LIN {X 0,Y 277.777,Z 1042.404,A -85,B 0,C 180,E1 8080.573,E2 8080.573} C_VEL
LIN {X 0,Y 260.235,Z 1059.705,A -85,B 0,C 180,E1 8078.402,E2 8078.402} C_VEL
LIN {X 0,Y 244.784,Z 1073.617,A -85,B 0,C 180,E1 8076.2,E2 8076.2} C_VEL
LIN {X 0,Y 227.244,Z 1088.097,A -85,B 0,C 180,E1 8073.276,E2 8073.276} C_VEL
LIN {X 0,Y 207.963,Z 1102.365,A -85,B 0,C 180,E1 8069.385,E2 8069.385} C_VEL
LIN {X 0,Y 192.676,Z 1112.751,A -85,B 0,C 180,E1 8065.598,E2 8065.598} C_VEL
LIN {X 0,Y 177.571,Z 1122.315,A -85,B 0,C 180,E1 8060.99,E2 8060.99} C_VEL
LIN {X 0,Y 159.969,Z 1132.7,A -85,B 0,C 180,E1 8053.93,E2 8053.93} C_VEL
LIN {X 0,Y 147.003,Z 1139.922,A -85,B 0,C 180,E1 8046.765,E2 8046.765} C_VEL
LIN {X 0,Y 137.193,Z 1145.374,A -85,B 0,C 180,E1 8039.228,E2 8039.228} C_VEL
LIN {X 0,Y 128.774,Z 1150.343,A -85,B 0,C 180,E1 8029.504,E2 8029.504} C_VEL
LIN {X 0,Y 123.283,Z 1154.147,A -85,B 0,C 180,E1 8017.925,E2 8017.925} C_VEL
LIN {X 0,Y 121.496,Z 1156.08,A -85,B 0,C 180,E1 8008.585,E2 8008.585} C_VEL
LIN {X 0,Y 121.206,Z 1157.152,A -85,B 0,C 180,E1 8000.024,E2 8000.024} C_VEL
LIN {X 0,Y 121.981,Z 1157.579,A -85,B 0,C 180,E1 7990.86,E2 7990.86} C_VEL
LIN {X 0,Y 124.84,Z 1157.139,A -85,B 0,C 180,E1 7980.754,E2 7980.754} C_VEL
LIN {X 0,Y 130.177,Z 1155.784,A -85,B 0,C 180,E1 7971.527,E2 7971.527} C_VEL
LIN {X 0,Y 138.594,Z 1153.323,A -85,B 0,C 180,E1 7962.62,E2 7962.62} C_VEL
LIN {X 0,Y 152.039,Z 1149.022,A -85,B 0,C 180,E1 7953.364,E2 7953.364} C_VEL
LIN {X 0,Y 168.555,Z 1142.861,A -85,B 0,C 180,E1 7945.623,E2 7945.623} C_VEL
LIN {X 0,Y 183.712,Z 1136.651,A -85,B 0,C 180,E1 7940.385,E2 7940.385} C_VEL
LIN {X 0,Y 201.418,Z 1128.646,A -85,B 0,C 180,E1 7935.627,E2 7935.627} C_VEL
LIN {X 0,Y 223.132,Z 1117.531,A -85,B 0,C 180,E1 7931.085,E2 7931.085} C_VEL
LIN {X 0,Y 241.336,Z 1107.052,A -85,B 0,C 180,E1 7928.035,E2 7928.035} C_VEL
LIN {X 0,Y 259.171,Z 1095.723,A -85,B 0,C 180,E1 7925.532,E2 7925.532} C_VEL
LIN {X 0,Y 280.353,Z 1080.74,A -85,B 0,C 180,E1 7923.031,E2 7923.031} C_VEL
LIN {X 0,Y 299.018,Z 1065.79,A -85,B 0,C 180,E1 7921.149,E2 7921.149} C_VEL
LIN {X 0,Y 314.959,Z 1051.738,A -85,B 0,C 180,E1 7919.738,E2 7919.738} C_VEL
LIN {X 0,Y 331.272,Z 1035.907,A -85,B 0,C 180,E1 7918.443,E2 7918.443} C_VEL
LIN {X 0,Y 336.652,Z 1030.337,A -85,B 0,C 180,E1 7918.031,E2 7918.031} C_VEL
LIN {X 0,Y 326.224,Z 1041.38,A -85,B 0,C 180,E1 7917.323,E2 7917.323} C_VEL
LIN {X 0,Y 320.827,Z 1046.926,A -85,B 0,C 180,E1 7917.12,E2 7917.12} C_VEL
LIN {X 0,Y 305.219,Z 1061.315,A -85,B 0,C 180,E1 7917.168,E2 7917.168} C_VEL
LIN {X 0,Y 300.311,Z 1065.535,A -85,B 0,C 180,E1 7916.938,E2 7916.938} C_VEL
LIN {X 0,Y 283.815,Z 1079.451,A -85,B 0,C 180,E1 7915.551,E2 7915.551} C_VEL
LIN {X 0,Y 264.581,Z 1094.292,A -85,B 0,C 180,E1 7913.66,E2 7913.66} C_VEL
LIN {X 0,Y 241.035,Z 1110.559,A -85,B 0,C 180,E1 7910.847,E2 7910.847} C_VEL
LIN {X 0,Y 222,Z 1122.424,A -85,B 0,C 180,E1 7908.043,E2 7908.043} C_VEL
LIN {X 0,Y 203.24,Z 1133.159,A -85,B 0,C 180,E1 7904.632,E2 7904.632} C_VEL
LIN {X 0,Y 180.343,Z 1145.085,A -85,B 0,C 180,E1 7899.216,E2 7899.216} C_VEL
LIN {X 0,Y 162.143,Z 1153.663,A -85,B 0,C 180,E1 7893.399,E2 7893.399} C_VEL
LIN {X 0,Y 146.993,Z 1160.411,A -85,B 0,C 180,E1 7886.789,E2 7886.789} C_VEL
LIN {X 0,Y 131.975,Z 1166.918,A -85,B 0,C 180,E1 7877.298,E2 7877.298} C_VEL
LIN {X 0,Y 120.616,Z 1171.822,A -85,B 0,C 180,E1 7865.47,E2 7865.47} C_VEL
LIN {X 0,Y 115.084,Z 1174.558,A -85,B 0,C 180,E1 7854.647,E2 7854.647} C_VEL
LIN {X 0,Y 113.015,Z 1175.991,A -85,B 0,C 180,E1 7844.867,E2 7844.867} C_VEL
LIN {X 0,Y 112.884,Z 1176.51,A -85,B 0,C 180,E1 7836.102,E2 7836.102} C_VEL
LIN {X 0,Y 113.083,Z 1176.346,A -85,B 0,C 180,E1 7829.494,E2 7829.494} C_VEL
LIN {X 0,Y 112.893,Z 1175.456,A -85,B 0,C 180,E1 7822.366,E2 7822.366} C_VEL
LIN {X 0,Y 113.288,Z 1173.656,A -85,B 0,C 180,E1 7813.595,E2 7813.595} C_VEL
LIN {X 0,Y 115.693,Z 1170.698,A -85,B 0,C 180,E1 7803.848,E2 7803.848} C_VEL
LIN {X 0,Y 120.925,Z 1166.519,A -85,B 0,C 180,E1 7794.052,E2 7794.052} C_VEL
LIN {X 0,Y 129.84,Z 1160.665,A -85,B 0,C 180,E1 7784.262,E2 7784.262} C_VEL
LIN {X 0,Y 144.741,Z 1151.55,A -85,B 0,C 180,E1 7774.009,E2 7774.009} C_VEL
LIN {X 0,Y 158.897,Z 1142.863,A -85,B 0,C 180,E1 7767.346,E2 7767.346} C_VEL
LIN {X 0,Y 173.719,Z 1133.462,A -85,B 0,C 180,E1 7762.082,E2 7762.082} C_VEL
LIN {X 0,Y 192.717,Z 1120.731,A -85,B 0,C 180,E1 7756.891,E2 7756.891} C_VEL
LIN {X 0,Y 212.206,Z 1106.31,A -85,B 0,C 180,E1 7752.755,E2 7752.755} C_VEL
LIN {X 0,Y 228.409,Z 1093.381,A -85,B 0,C 180,E1 7749.96,E2 7749.96} C_VEL
LIN {X 0,Y 246.957,Z 1077.339,A -85,B 0,C 180,E1 7747.284,E2 7747.284} C_VEL
LIN {X 0,Y 266.154,Z 1058.803,A -85,B 0,C 180,E1 7744.957,E2 7744.957} C_VEL
LIN {X 0,Y 281.444,Z 1042.59,A -85,B 0,C 180,E1 7743.365,E2 7743.365} C_VEL
LIN {X 0,Y 296.14,Z 1025.559,A -85,B 0,C 180,E1 7742.016,E2 7742.016} C_VEL
LIN {X 0,Y 313.472,Z 1003.187,A -85,B 0,C 180,E1 7740.603,E2 7740.603} C_VEL
LIN {X 0,Y 326.96,Z 983.532,A -85,B 0,C 180,E1 7739.615,E2 7739.615} C_VEL
LIN {X 0,Y 338.52,Z 964.867,A -85,B 0,C 180,E1 7738.848,E2 7738.848} C_VEL
LIN {X 0,Y 350.134,Z 943.92,A -85,B 0,C 180,E1 7738.141,E2 7738.141} C_VEL
LIN {X 0,Y 362.303,Z 918.548,A -85,B 0,C 180,E1 7737.463,E2 7737.463} C_VEL
LIN {X 0,Y 371.204,Z 896.845,A -85,B 0,C 180,E1 7737.002,E2 7737.002} C_VEL
LIN {X 0,Y 378.593,Z 875.937,A -85,B 0,C 180,E1 7736.647,E2 7736.647} C_VEL
LIN {X 0,Y 386.321,Z 849.767,A -85,B 0,C 180,E1 7736.294,E2 7736.294} C_VEL
LIN {X 0,Y 392.167,Z 823.299,A -85,B 0,C 180,E1 7735.962,E2 7735.962} C_VEL
LIN {X 0,Y 395.874,Z 800.827,A -85,B 0,C 180,E1 7735.692,E2 7735.692} C_VEL
LIN {X 0,Y 411.944,Z 668.915,A -85,B 0,C 180,E1 7734.149,E2 7734.149} C_VEL
LIN {X 0,Y 411.886,Z 668.578,A -85,B 0,C 180,E1 7732.827,E2 7732.827} C_VEL
LIN {X 0,Y 395.068,Z 804.017,A -85,B 0,C 180,E1 7731.344,E2 7731.344} C_VEL
LIN {X 0,Y 390.125,Z 831.221,A -85,B 0,C 180,E1 7731.017,E2 7731.017} C_VEL
LIN {X 0,Y 383.915,Z 855.88,A -85,B 0,C 180,E1 7730.656,E2 7730.656} C_VEL
LIN {X 0,Y 377.386,Z 877.053,A -85,B 0,C 180,E1 7730.26,E2 7730.26} C_VEL
LIN {X 0,Y 369.182,Z 899.494,A -85,B 0,C 180,E1 7729.75,E2 7729.75} C_VEL
LIN {X 0,Y 357.977,Z 925.058,A -85,B 0,C 180,E1 7729.041,E2 7729.041} C_VEL
LIN {X 0,Y 347.61,Z 945.408,A -85,B 0,C 180,E1 7728.351,E2 7728.351} C_VEL
LIN {X 0,Y 336.359,Z 964.986,A -85,B 0,C 180,E1 7727.553,E2 7727.553} C_VEL
LIN {X 0,Y 320.984,Z 988.506,A -85,B 0,C 180,E1 7726.378,E2 7726.378} C_VEL
LIN {X 0,Y 307.112,Z 1007.162,A -85,B 0,C 180,E1 7725.225,E2 7725.225} C_VEL
LIN {X 0,Y 293.331,Z 1023.926,A -85,B 0,C 180,E1 7723.972,E2 7723.972} C_VEL
LIN {X 0,Y 276.154,Z 1042.849,A -85,B 0,C 180,E1 7722.219,E2 7722.219} C_VEL
LIN {X 0,Y 258.315,Z 1060.173,A -85,B 0,C 180,E1 7720.149,E2 7720.149} C_VEL
LIN {X 0,Y 242.565,Z 1074.107,A -85,B 0,C 180,E1 7718.041,E2 7718.041} C_VEL
LIN {X 0,Y 225.211,Z 1088.146,A -85,B 0,C 180,E1 7715.333,E2 7715.333} C_VEL
LIN {X 0,Y 205.644,Z 1102.352,A -85,B 0,C 180,E1 7711.646,E2 7711.646} C_VEL
LIN {X 0,Y 189.064,Z 1113.295,A -85,B 0,C 180,E1 7707.795,E2 7707.795} C_VEL
LIN {X 0,Y 173.391,Z 1122.869,A -85,B 0,C 180,E1 7703.277,E2 7703.277} C_VEL
LIN {X 0,Y 154.965,Z 1133.274,A -85,B 0,C 180,E1 7696.273,E2 7696.273} C_VEL
LIN {X 0,Y 141.245,Z 1140.508,A -85,B 0,C 180,E1 7689.051,E2 7689.051} C_VEL
LIN {X 0,Y 130.741,Z 1145.97,A -85,B 0,C 180,E1 7681.334,E2 7681.334} C_VEL
LIN {X 0,Y 121.602,Z 1150.949,A -85,B 0,C 180,E1 7671.21,E2 7671.21} C_VEL
LIN {X 0,Y 115.555,Z 1154.773,A -85,B 0,C 180,E1 7658.96,E2 7658.96} C_VEL
LIN {X 0,Y 113.555,Z 1156.718,A -85,B 0,C 180,E1 7648.991,E2 7648.991} C_VEL
LIN {X 0,Y 113.228,Z 1157.773,A -85,B 0,C 180,E1 7640.341,E2 7640.341} C_VEL
LIN {X 0,Y 114.037,Z 1158.259,A -85,B 0,C 180,E1 7630.538,E2 7630.538} C_VEL
LIN {X 0,Y 117.279,Z 1157.848,A -85,B 0,C 180,E1 7619.441,E2 7619.441} C_VEL
LIN {X 0,Y 123.277,Z 1156.494,A -85,B 0,C 180,E1 7609.544,E2 7609.544} C_VEL
LIN {X 0,Y 132.45,Z 1154.053,A -85,B 0,C 180,E1 7600.32,E2 7600.32} C_VEL
LIN {X 0,Y 146.847,Z 1149.768,A -85,B 0,C 180,E1 7590.917,E2 7590.917} C_VEL
LIN {X 0,Y 164.266,Z 1143.642,A -85,B 0,C 180,E1 7583.203,E2 7583.203} C_VEL
LIN {X 0,Y 180.708,Z 1137.198,A -85,B 0,C 180,E1 7577.884,E2 7577.884} C_VEL
LIN {X 0,Y 199.275,Z 1129.085,A -85,B 0,C 180,E1 7573.247,E2 7573.247} C_VEL
LIN {X 0,Y 221.644,Z 1117.902,A -85,B 0,C 180,E1 7568.909,E2 7568.909} C_VEL
LIN {X 0,Y 239.344,Z 1107.948,A -85,B 0,C 180,E1 7566.151,E2 7566.151} C_VEL
LIN {X 0,Y 257.36,Z 1096.75,A -85,B 0,C 180,E1 7563.787,E2 7563.787} C_VEL
LIN {X 0,Y 278.636,Z 1082.047,A -85,B 0,C 180,E1 7561.439,E2 7561.439} C_VEL
LIN {X 0,Y 297.998,Z 1066.806,A -85,B 0,C 180,E1 7559.615,E2 7559.615} C_VEL
LIN {X 0,Y 314.096,Z 1052.824,A -85,B 0,C 180,E1 7558.287,E2 7558.287} C_VEL
LIN {X 0,Y 316.126,Z 1050.98,A -85,B 0,C 180,E1 7558.116,E2 7558.116} C_VEL
LIN {X 0,Y 300.311,Z 1065.535,A -85,B 0,C 180,E1 7556.938,E2 7556.938} C_VEL
LIN {X 0,Y 294.497,Z 1070.582,A -85,B 0,C 180,E1 7556.674,E2 7556.674} C_VEL
LIN {X 0,Y 277.819,Z 1083.663,A -85,B 0,C 180,E1 7556.596,E2 7556.596} C_VEL
LIN {X 0,Y 272.61,Z 1087.499,A -85,B 0,C 180,E1 7556.3,E2 7556.3} C_VEL
LIN {X 0,Y 254.145,Z 1100.73,A -85,B 0,C 180,E1 7554.476,E2 7554.476} C_VEL
LIN {X 0,Y 236.061,Z 1112.577,A -85,B 0,C 180,E1 7552.363,E2 7552.363} C_VEL
LIN {X 0,Y 214.7,Z 1125.373,A -85,B 0,C 180,E1 7549.305,E2 7549.305} C_VEL
LIN {X 0,Y 191.472,Z 1137.745,A -85,B 0,C 180,E1 7545.031,E2 7545.031} C_VEL
LIN {X 0,Y 172.839,Z 1146.738,A -85,B 0,C 180,E1 7540.552,E2 7540.552} C_VEL
LIN {X 0,Y 155.475,Z 1154.467,A -85,B 0,C 180,E1 7535.063,E2 7535.063} C_VEL
LIN {X 0,Y 135.912,Z 1162.579,A -85,B 0,C 180,E1 7526.233,E2 7526.233} C_VEL
LIN {X 0,Y 121.7,Z 1168.098,A -85,B 0,C 180,E1 7516.302,E2 7516.302} C_VEL
LIN {X 0,Y 112.609,Z 1171.717,A -85,B 0,C 180,E1 7506.097,E2 7506.097} C_VEL
LIN {X 0,Y 107.146,Z 1174.147,A -85,B 0,C 180,E1 7495.148,E2 7495.148} C_VEL
LIN {X 0,Y 105.029,Z 1175.421,A -85,B 0,C 180,E1 7484.895,E2 7484.895} C_VEL
LIN {X 0,Y 104.915,Z 1175.827,A -85,B 0,C 180,E1 7476.018,E2 7476.018} C_VEL
LIN {X 0,Y 105.101,Z 1175.656,A -85,B 0,C 180,E1 7468.91,E2 7468.91} C_VEL
LIN {X 0,Y 104.894,Z 1174.675,A -85,B 0,C 180,E1 7461.228,E2 7461.228} C_VEL
LIN {X 0,Y 105.743,Z 1172.522,A -85,B 0,C 180,E1 7450.674,E2 7450.674} C_VEL
LIN {X 0,Y 110.604,Z 1168.253,A -85,B 0,C 180,E1 7437.153,E2 7437.153} C_VEL
LIN {X 0,Y 120.125,Z 1162.081,A -85,B 0,C 180,E1 7424.969,E2 7424.969} C_VEL
LIN {X 0,Y 130.733,Z 1155.946,A -85,B 0,C 180,E1 7416.578,E2 7416.578} C_VEL
LIN {X 0,Y 143.528,Z 1148.661,A -85,B 0,C 180,E1 7409.451,E2 7409.451} C_VEL
LIN {X 0,Y 161.134,Z 1138.402,A -85,B 0,C 180,E1 7402.398,E2 7402.398} C_VEL
LIN {X 0,Y 180.613,Z 1126.073,A -85,B 0,C 180,E1 7396.723,E2 7396.723} C_VEL
LIN {X 0,Y 197.028,Z 1114.923,A -85,B 0,C 180,E1 7393.008,E2 7393.008} C_VEL
LIN {X 0,Y 214.129,Z 1102.4,A -85,B 0,C 180,E1 7389.856,E2 7389.856} C_VEL
LIN {X 0,Y 236.156,Z 1084.612,A -85,B 0,C 180,E1 7386.564,E2 7386.564} C_VEL
LIN {X 0,Y 252.747,Z 1069.774,A -85,B 0,C 180,E1 7384.513,E2 7384.513} C_VEL
LIN {X 0,Y 268.292,Z 1054.632,A -85,B 0,C 180,E1 7382.845,E2 7382.845} C_VEL
LIN {X 0,Y 286.516,Z 1035.175,A -85,B 0,C 180,E1 7381.153,E2 7381.153} C_VEL
LIN {X 0,Y 303.408,Z 1014.71,A -85,B 0,C 180,E1 7379.78,E2 7379.78} C_VEL
LIN {X 0,Y 317.023,Z 996.487,A -85,B 0,C 180,E1 7378.802,E2 7378.802} C_VEL
LIN {X 0,Y 331.178,Z 975.452,A -85,B 0,C 180,E1 7377.88,E2 7377.88} C_VEL
LIN {X 0,Y 345.41,Z 951.169,A -85,B 0,C 180,E1 7377.043,E2 7377.043} C_VEL
LIN {X 0,Y 355.613,Z 931.378,A -85,B 0,C 180,E1 7376.495,E2 7376.495} C_VEL
LIN {X 0,Y 364.819,Z 911.173,A -85,B 0,C 180,E1 7376.039,E2 7376.039} C_VEL
LIN {X 0,Y 374.81,Z 885.761,A -85,B 0,C 180,E1 7375.58,E2 7375.58} C_VEL
LIN {X 0,Y 382.862,Z 860.41,A -85,B 0,C 180,E1 7375.234,E2 7375.234} C_VEL
LIN {X 0,Y 388.579,Z 838.407,A -85,B 0,C 180,E1 7374.972,E2 7374.972} C_VEL
LIN {X 0,Y 394.017,Z 811.54,A -85,B 0,C 180,E1 7374.653,E2 7374.653} C_VEL
LIN {X 0,Y 400.006,Z 765.699,A -85,B 0,C 180,E1 7374.134,E2 7374.134} C_VEL
LIN {X 0,Y 406.812,Z 709.958,A -85,B 0,C 180,E1 7373.507,E2 7373.507} C_VEL
LIN {X 0,Y 394.778,Z 805.105,A -85,B 0,C 180,E1 7372.496,E2 7372.496} C_VEL
LIN {X 0,Y 389.482,Z 833.336,A -85,B 0,C 180,E1 7372.17,E2 7372.17} C_VEL
LIN {X 0,Y 383.513,Z 856.711,A -85,B 0,C 180,E1 7371.842,E2 7371.842} C_VEL
LIN {X 0,Y 376.858,Z 878.056,A -85,B 0,C 180,E1 7371.463,E2 7371.463} C_VEL
LIN {X 0,Y 368.031,Z 901.872,A -85,B 0,C 180,E1 7370.947,E2 7370.947} C_VEL
LIN {X 0,Y 357.056,Z 926.357,A -85,B 0,C 180,E1 7370.298,E2 7370.298} C_VEL
LIN {X 0,Y 346.595,Z 946.622,A -85,B 0,C 180,E1 7369.646,E2 7369.646} C_VEL
LIN {X 0,Y 334.762,Z 966.913,A -85,B 0,C 180,E1 7368.858,E2 7368.858} C_VEL
LIN {X 0,Y 319.229,Z 990.185,A -85,B 0,C 180,E1 7367.745,E2 7367.745} C_VEL
LIN {X 0,Y 305.67,Z 1008.156,A -85,B 0,C 180,E1 7366.688,E2 7366.688} C_VEL
LIN {X 0,Y 291.966,Z 1024.6,A -85,B 0,C 180,E1 7365.522,E2 7365.522} C_VEL
LIN {X 0,Y 274.761,Z 1043.293,A -85,B 0,C 180,E1 7363.883,E2 7363.883} C_VEL
LIN {X 0,Y 256.638,Z 1060.638,A -85,B 0,C 180,E1 7361.919,E2 7361.919} C_VEL
LIN {X 0,Y 240.601,Z 1074.586,A -85,B 0,C 180,E1 7359.914,E2 7359.914} C_VEL
LIN {X 0,Y 223.146,Z 1088.435,A -85,B 0,C 180,E1 7357.372,E2 7357.372} C_VEL
LIN {X 0,Y 202.822,Z 1102.883,A -85,B 0,C 180,E1 7353.793,E2 7353.793} C_VEL
LIN {X 0,Y 185.741,Z 1113.838,A -85,B 0,C 180,E1 7350.074,E2 7350.074} C_VEL
LIN {X 0,Y 169.5,Z 1123.424,A -85,B 0,C 180,E1 7345.674,E2 7345.674} C_VEL
LIN {X 0,Y 150.236,Z 1133.849,A -85,B 0,C 180,E1 7338.767,E2 7338.767} C_VEL
LIN {X 0,Y 135.731,Z 1141.093,A -85,B 0,C 180,E1 7331.527,E2 7331.527} C_VEL
LIN {X 0,Y 124.003,Z 1146.804,A -85,B 0,C 180,E1 7323.25,E2 7323.25} C_VEL
LIN {X 0,Y 113.559,Z 1152.134,A -85,B 0,C 180,E1 7311.703,E2 7311.703} C_VEL
LIN {X 0,Y 107.523,Z 1155.613,A -85,B 0,C 180,E1 7299.095,E2 7299.095} C_VEL
LIN {X 0,Y 105.564,Z 1157.421,A -85,B 0,C 180,E1 7288.914,E2 7288.914} C_VEL
LIN {X 0,Y 105.263,Z 1158.454,A -85,B 0,C 180,E1 7279.602,E2 7279.602} C_VEL
LIN {X 0,Y 106.286,Z 1158.922,A -85,B 0,C 180,E1 7269.055,E2 7269.055} C_VEL
LIN {X 0,Y 109.968,Z 1158.522,A -85,B 0,C 180,E1 7257.558,E2 7257.558} C_VEL
LIN {X 0,Y 116.947,Z 1157.112,A -85,B 0,C 180,E1 7246.845,E2 7246.845} C_VEL
LIN {X 0,Y 127.299,Z 1154.59,A -85,B 0,C 180,E1 7237.215,E2 7237.215} C_VEL
LIN {X 0,Y 143.315,Z 1150.101,A -85,B 0,C 180,E1 7227.621,E2 7227.621} C_VEL
LIN {X 0,Y 161.3,Z 1144.062,A -85,B 0,C 180,E1 7220.313,E2 7220.313} C_VEL
LIN {X 0,Y 178.255,Z 1137.669,A -85,B 0,C 180,E1 7215.253,E2 7215.253} C_VEL
LIN {X 0,Y 199.644,Z 1128.59,A -85,B 0,C 180,E1 7210.387,E2 7210.387} C_VEL
LIN {X 0,Y 221.42,Z 1117.773,A -85,B 0,C 180,E1 7206.562,E2 7206.562} C_VEL
LIN {X 0,Y 239.545,Z 1107.723,A -85,B 0,C 180,E1 7203.983,E2 7203.983} C_VEL
LIN {X 0,Y 260.139,Z 1095.029,A -85,B 0,C 180,E1 7201.542,E2 7201.542} C_VEL
LIN {X 0,Y 281.977,Z 1079.686,A -85,B 0,C 180,E1 7199.375,E2 7199.375} C_VEL
LIN {X 0,Y 295.48,Z 1069.244,A -85,B 0,C 180,E1 7198.191,E2 7198.191} C_VEL
LIN {X 0,Y 272.61,Z 1087.499,A -85,B 0,C 180,E1 7196.3,E2 7196.3} C_VEL
LIN {X 0,Y 266.443,Z 1091.967,A -85,B 0,C 180,E1 7195.957,E2 7195.957} C_VEL
LIN {X 0,Y 248.815,Z 1103.729,A -85,B 0,C 180,E1 7195.707,E2 7195.707} C_VEL
LIN {X 0,Y 243.349,Z 1107.141,A -85,B 0,C 180,E1 7195.325,E2 7195.325} C_VEL
LIN {X 0,Y 221.751,Z 1120.145,A -85,B 0,C 180,E1 7192.732,E2 7192.732} C_VEL
LIN {X 0,Y 202.164,Z 1130.863,A -85,B 0,C 180,E1 7189.805,E2 7189.805} C_VEL
LIN {X 0,Y 179.7,Z 1142.025,A -85,B 0,C 180,E1 7185.499,E2 7185.499} C_VEL
LIN {X 0,Y 157.71,Z 1151.642,A -85,B 0,C 180,E1 7179.768,E2 7179.768} C_VEL
LIN {X 0,Y 140.616,Z 1158.47,A -85,B 0,C 180,E1 7173.629,E2 7173.629} C_VEL
LIN {X 0,Y 125.469,Z 1164.126,A -85,B 0,C 180,E1 7165.973,E2 7165.973} C_VEL
LIN {X 0,Y 110.496,Z 1169.569,A -85,B 0,C 180,E1 7154.168,E2 7154.168} C_VEL
LIN {X 0,Y 101.015,Z 1172.988,A -85,B 0,C 180,E1 7140.319,E2 7140.319} C_VEL
LIN {X 0,Y 97.401,Z 1174.623,A -85,B 0,C 180,E1 7127.937,E2 7127.937} C_VEL
LIN {X 0,Y 96.899,Z 1175.155,A -85,B 0,C 180,E1 7117.113,E2 7117.113} C_VEL
LIN {X 0,Y 97.145,Z 1175.024,A -85,B 0,C 180,E1 7110,E2 7110} C_VEL
LIN {X 0,Y 96.936,Z 1174.199,A -85,B 0,C 180,E1 7102.294,E2 7102.294} C_VEL
LIN {X 0,Y 97.402,Z 1172.557,A -85,B 0,C 180,E1 7092.681,E2 7092.681} C_VEL
LIN {X 0,Y 100.414,Z 1169.604,A -85,B 0,C 180,E1 7081.196,E2 7081.196} C_VEL
LIN {X 0,Y 106.679,Z 1165.509,A -85,B 0,C 180,E1 7070.227,E2 7070.227} C_VEL
LIN {X 0,Y 116.424,Z 1160.078,A -85,B 0,C 180,E1 7060.153,E2 7060.153} C_VEL
LIN {X 0,Y 132.008,Z 1151.873,A -85,B 0,C 180,E1 7049.995,E2 7049.995} C_VEL
LIN {X 0,Y 150.104,Z 1141.865,A -85,B 0,C 180,E1 7042.197,E2 7042.197} C_VEL
LIN {X 0,Y 166.331,Z 1132.42,A -85,B 0,C 180,E1 7037.101,E2 7037.101} C_VEL
LIN {X 0,Y 186.268,Z 1119.964,A -85,B 0,C 180,E1 7032.327,E2 7032.327} C_VEL
LIN {X 0,Y 206.294,Z 1106.019,A -85,B 0,C 180,E1 7028.609,E2 7028.609} C_VEL
LIN {X 0,Y 223.213,Z 1093.186,A -85,B 0,C 180,E1 7026.056,E2 7026.056} C_VEL
LIN {X 0,Y 239.541,Z 1079.727,A -85,B 0,C 180,E1 7023.974,E2 7023.974} C_VEL
LIN {X 0,Y 259.099,Z 1062.095,A -85,B 0,C 180,E1 7021.864,E2 7021.864} C_VEL
LIN {X 0,Y 277.152,Z 1043.73,A -85,B 0,C 180,E1 7020.207,E2 7020.207} C_VEL
LIN {X 0,Y 292.005,Z 1027.135,A -85,B 0,C 180,E1 7019.019,E2 7019.019} C_VEL
LIN {X 0,Y 306.142,Z 1009.764,A -85,B 0,C 180,E1 7018.001,E2 7018.001} C_VEL
LIN {X 0,Y 322.918,Z 986.713,A -85,B 0,C 180,E1 7016.925,E2 7016.925} C_VEL
LIN {X 0,Y 336.365,Z 965.64,A -85,B 0,C 180,E1 7016.153,E2 7016.153} C_VEL
LIN {X 0,Y 347.488,Z 946.12,A -85,B 0,C 180,E1 7015.571,E2 7015.571} C_VEL
LIN {X 0,Y 359.661,Z 921.926,A -85,B 0,C 180,E1 7014.993,E2 7014.993} C_VEL
LIN {X 0,Y 370.133,Z 897.031,A -85,B 0,C 180,E1 7014.528,E2 7014.528} C_VEL
LIN {X 0,Y 377.617,Z 876.276,A -85,B 0,C 180,E1 7014.225,E2 7014.225} C_VEL
LIN {X 0,Y 384.765,Z 852.709,A -85,B 0,C 180,E1 7013.949,E2 7013.949} C_VEL
LIN {X 0,Y 391.358,Z 824.544,A -85,B 0,C 180,E1 7013.632,E2 7013.632} C_VEL
LIN {X 0,Y 392.801,Z 817.005,A -85,B 0,C 180,E1 7013.538,E2 7013.538} C_VEL
LIN {X 0,Y 387.96,Z 839.737,A -85,B 0,C 180,E1 7013.272,E2 7013.272} C_VEL
LIN {X 0,Y 382.246,Z 861.074,A -85,B 0,C 180,E1 7012.974,E2 7012.974} C_VEL
LIN {X 0,Y 373.54,Z 887.479,A -85,B 0,C 180,E1 7012.513,E2 7012.513} C_VEL
LIN {X 0,Y 363.995,Z 911.017,A -85,B 0,C 180,E1 7011.995,E2 7011.995} C_VEL
LIN {X 0,Y 354.868,Z 930.54,A -85,B 0,C 180,E1 7011.478,E2 7011.478} C_VEL
LIN {X 0,Y 343.367,Z 952.168,A -85,B 0,C 180,E1 7010.801,E2 7010.801} C_VEL
LIN {X 0,Y 329.05,Z 975.411,A -85,B 0,C 180,E1 7009.902,E2 7009.902} C_VEL
LIN {X 0,Y 316.235,Z 993.795,A -85,B 0,C 180,E1 7009.028,E2 7009.028} C_VEL
LIN {X 0,Y 303.019,Z 1010.904,A -85,B 0,C 180,E1 7008.055,E2 7008.055} C_VEL
LIN {X 0,Y 285.687,Z 1031.08,A -85,B 0,C 180,E1 7006.644,E2 7006.644} C_VEL
LIN {X 0,Y 268.059,Z 1049.088,A -85,B 0,C 180,E1 7005.031,E2 7005.031} C_VEL
LIN {X 0,Y 252.474,Z 1063.531,A -85,B 0,C 180,E1 7003.41,E2 7003.41} C_VEL
LIN {X 0,Y 234.416,Z 1078.746,A -85,B 0,C 180,E1 7001.244,E2 7001.244} C_VEL
LIN {X 0,Y 214.089,Z 1093.975,A -85,B 0,C 180,E1 6998.339,E2 6998.339} C_VEL
LIN {X 0,Y 196.895,Z 1105.581,A -85,B 0,C 180,E1 6995.365,E2 6995.365} C_VEL
LIN {X 0,Y 179.46,Z 1116.328,A -85,B 0,C 180,E1 6991.677,E2 6991.677} C_VEL
LIN {X 0,Y 158.247,Z 1128.094,A -85,B 0,C 180,E1 6985.863,E2 6985.863} C_VEL
LIN {X 0,Y 142.32,Z 1136.084,A -85,B 0,C 180,E1 6979.975,E2 6979.975} C_VEL
LIN {X 0,Y 128.644,Z 1142.533,A -85,B 0,C 180,E1 6973.153,E2 6973.153} C_VEL
LIN {X 0,Y 114.946,Z 1148.831,A -85,B 0,C 180,E1 6963.23,E2 6963.23} C_VEL
LIN {X 0,Y 104.537,Z 1153.646,A -85,B 0,C 180,E1 6950.725,E2 6950.725} C_VEL
LIN {X 0,Y 99.492,Z 1156.452,A -85,B 0,C 180,E1 6939.253,E2 6939.253} C_VEL
LIN {X 0,Y 97.571,Z 1158.125,A -85,B 0,C 180,E1 6928.825,E2 6928.825} C_VEL
LIN {X 0,Y 97.293,Z 1159.105,A -85,B 0,C 180,E1 6919.34,E2 6919.34} C_VEL
LIN {X 0,Y 98.369,Z 1159.601,A -85,B 0,C 180,E1 6908.535,E2 6908.535} C_VEL
LIN {X 0,Y 102.682,Z 1159.214,A -85,B 0,C 180,E1 6895.613,E2 6895.613} C_VEL
LIN {X 0,Y 110.444,Z 1157.825,A -85,B 0,C 180,E1 6884.341,E2 6884.341} C_VEL
LIN {X 0,Y 121.486,Z 1155.373,A -85,B 0,C 180,E1 6874.604,E2 6874.604} C_VEL
LIN {X 0,Y 138.081,Z 1151.08,A -85,B 0,C 180,E1 6865.157,E2 6865.157} C_VEL
LIN {X 0,Y 157.459,Z 1144.932,A -85,B 0,C 180,E1 6857.732,E2 6857.732} C_VEL
LIN {X 0,Y 175.309,Z 1138.476,A -85,B 0,C 180,E1 6852.766,E2 6852.766} C_VEL
LIN {X 0,Y 195.129,Z 1130.351,A -85,B 0,C 180,E1 6848.525,E2 6848.525} C_VEL
LIN {X 0,Y 218.683,Z 1119.145,A -85,B 0,C 180,E1 6844.63,E2 6844.63} C_VEL
LIN {X 0,Y 238.121,Z 1108.625,A -85,B 0,C 180,E1 6842.061,E2 6842.061} C_VEL
LIN {X 0,Y 256.964,Z 1097.266,A -85,B 0,C 180,E1 6839.976,E2 6839.976} C_VEL
LIN {X 0,Y 274.857,Z 1085.292,A -85,B 0,C 180,E1 6838.275,E2 6838.275} C_VEL
LIN {X 0,Y 254.448,Z 1099.765,A -85,B 0,C 180,E1 6836.465,E2 6836.465} C_VEL
LIN {X 0,Y 243.349,Z 1107.141,A -85,B 0,C 180,E1 6835.325,E2 6835.325} C_VEL
LIN {X 0,Y 236.859,Z 1111.078,A -85,B 0,C 180,E1 6834.875,E2 6834.875} C_VEL
LIN {X 0,Y 219.3,Z 1120.772,A -85,B 0,C 180,E1 6834.44,E2 6834.44} C_VEL
LIN {X 0,Y 212.766,Z 1124.284,A -85,B 0,C 180,E1 6833.882,E2 6833.882} C_VEL
LIN {X 0,Y 188.723,Z 1136.406,A -85,B 0,C 180,E1 6830.208,E2 6830.208} C_VEL
LIN {X 0,Y 168.828,Z 1145.39,A -85,B 0,C 180,E1 6826.232,E2 6826.232} C_VEL
LIN {X 0,Y 149.112,Z 1153.442,A -85,B 0,C 180,E1 6820.991,E2 6820.991} C_VEL
LIN {X 0,Y 125.832,Z 1161.906,A -85,B 0,C 180,E1 6811.885,E2 6811.885} C_VEL
LIN {X 0,Y 110.724,Z 1166.901,A -85,B 0,C 180,E1 6802.624,E2 6802.624} C_VEL
LIN {X 0,Y 99.42,Z 1170.524,A -85,B 0,C 180,E1 6791.588,E2 6791.588} C_VEL
LIN {X 0,Y 92.042,Z 1173.008,A -85,B 0,C 180,E1 6778.554,E2 6778.554} C_VEL
LIN {X 0,Y 89.006,Z 1174.326,A -85,B 0,C 180,E1 6764.309,E2 6764.309} C_VEL
LIN {X 0,Y 89.05,Z 1174.432,A -85,B 0,C 180,E1 6753.863,E2 6753.863} C_VEL
LIN {X 0,Y 89.12,Z 1174.154,A -85,B 0,C 180,E1 6747.428,E2 6747.428} C_VEL
LIN {X 0,Y 88.974,Z 1173.019,A -85,B 0,C 180,E1 6737.672,E2 6737.672} C_VEL
LIN {X 0,Y 91.438,Z 1170.159,A -85,B 0,C 180,E1 6723.364,E2 6723.364} C_VEL
LIN {X 0,Y 98.551,Z 1165.677,A -85,B 0,C 180,E1 6709.51,E2 6709.51} C_VEL
LIN {X 0,Y 108.843,Z 1160.353,A -85,B 0,C 180,E1 6698.659,E2 6698.659} C_VEL
LIN {X 0,Y 121.367,Z 1154.145,A -85,B 0,C 180,E1 6690.115,E2 6690.115} C_VEL
LIN {X 0,Y 137.485,Z 1146.001,A -85,B 0,C 180,E1 6682.542,E2 6682.542} C_VEL
LIN {X 0,Y 158.824,Z 1134.392,A -85,B 0,C 180,E1 6675.594,E2 6675.594} C_VEL
LIN {X 0,Y 176.437,Z 1123.921,A -85,B 0,C 180,E1 6671.37,E2 6671.37} C_VEL
LIN {X 0,Y 193.882,Z 1112.672,A -85,B 0,C 180,E1 6668.049,E2 6668.049} C_VEL
LIN {X 0,Y 215.278,Z 1097.567,A -85,B 0,C 180,E1 6664.796,E2 6664.796} C_VEL
LIN {X 0,Y 235.164,Z 1081.746,A -85,B 0,C 180,E1 6662.354,E2 6662.354} C_VEL
LIN {X 0,Y 251.978,Z 1067.089,A -85,B 0,C 180,E1 6660.621,E2 6660.621} C_VEL
LIN {X 0,Y 269.999,Z 1049.849,A -85,B 0,C 180,E1 6659.03,E2 6659.03} C_VEL
LIN {X 0,Y 288.481,Z 1029.945,A -85,B 0,C 180,E1 6657.616,E2 6657.616} C_VEL
LIN {X 0,Y 302.978,Z 1012.588,A -85,B 0,C 180,E1 6656.636,E2 6656.636} C_VEL
LIN {X 0,Y 316.805,Z 994.324,A -85,B 0,C 180,E1 6655.8,E2 6655.8} C_VEL
LIN {X 0,Y 332.233,Z 971.544,A -85,B 0,C 180,E1 6654.967,E2 6654.967} C_VEL
LIN {X 0,Y 345.137,Z 949.585,A -85,B 0,C 180,E1 6654.332,E2 6654.332} C_VEL
LIN {X 0,Y 355.58,Z 929.533,A -85,B 0,C 180,E1 6653.866,E2 6653.866} C_VEL
LIN {X 0,Y 365.838,Z 907.092,A -85,B 0,C 180,E1 6653.447,E2 6653.447} C_VEL
LIN {X 0,Y 366.885,Z 904.702,A -85,B 0,C 180,E1 6653.407,E2 6653.407} C_VEL
LIN {X 0,Y 356.214,Z 927.921,A -85,B 0,C 180,E1 6652.856,E2 6652.856} C_VEL
LIN {X 0,Y 346.063,Z 947.27,A -85,B 0,C 180,E1 6652.309,E2 6652.309} C_VEL
LIN {X 0,Y 334.501,Z 966.829,A -85,B 0,C 180,E1 6651.646,E2 6651.646} C_VEL
LIN {X 0,Y 318.667,Z 990.318,A -85,B 0,C 180,E1 6650.673,E2 6650.673} C_VEL
LIN {X 0,Y 304.343,Z 1008.972,A -85,B 0,C 180,E1 6649.719,E2 6649.719} C_VEL
LIN {X 0,Y 289.897,Z 1025.93,A -85,B 0,C 180,E1 6648.662,E2 6648.662} C_VEL
LIN {X 0,Y 271.745,Z 1045.094,A -85,B 0,C 180,E1 6647.171,E2 6647.171} C_VEL
LIN {X 0,Y 253.107,Z 1062.374,A -85,B 0,C 180,E1 6645.427,E2 6645.427} C_VEL
LIN {X 0,Y 236.549,Z 1076.28,A -85,B 0,C 180,E1 6643.636,E2 6643.636} C_VEL
LIN {X 0,Y 216.646,Z 1091.425,A -85,B 0,C 180,E1 6641.104,E2 6641.104} C_VEL
LIN {X 0,Y 196.322,Z 1105.01,A -85,B 0,C 180,E1 6637.958,E2 6637.958} C_VEL
LIN {X 0,Y 179.178,Z 1115.396,A -85,B 0,C 180,E1 6634.689,E2 6634.689} C_VEL
LIN {X 0,Y 161.058,Z 1125.391,A -85,B 0,C 180,E1 6630.357,E2 6630.357} C_VEL
LIN {X 0,Y 140.241,Z 1135.664,A -85,B 0,C 180,E1 6623.672,E2 6623.672} C_VEL
LIN {X 0,Y 124.902,Z 1142.552,A -85,B 0,C 180,E1 6616.758,E2 6616.758} C_VEL
LIN {X 0,Y 111.564,Z 1148.238,A -85,B 0,C 180,E1 6608.198,E2 6608.198} C_VEL
LIN {X 0,Y 99.312,Z 1153.526,A -85,B 0,C 180,E1 6595.652,E2 6595.652} C_VEL
LIN {X 0,Y 92.021,Z 1156.972,A -85,B 0,C 180,E1 6581.278,E2 6581.278} C_VEL
LIN {X 0,Y 89.636,Z 1158.762,A -85,B 0,C 180,E1 6569.36,E2 6569.36} C_VEL
LIN {X 0,Y 89.324,Z 1159.756,A -85,B 0,C 180,E1 6559.03,E2 6559.03} C_VEL
LIN {X 0,Y 90.587,Z 1160.273,A -85,B 0,C 180,E1 6547.274,E2 6547.274} C_VEL
LIN {X 0,Y 95.529,Z 1159.908,A -85,B 0,C 180,E1 6533.373,E2 6533.373} C_VEL
LIN {X 0,Y 104.285,Z 1158.517,A -85,B 0,C 180,E1 6521.421,E2 6521.421} C_VEL
LIN {X 0,Y 116.835,Z 1155.968,A -85,B 0,C 180,E1 6511.153,E2 6511.153} C_VEL
LIN {X 0,Y 135.425,Z 1151.403,A -85,B 0,C 180,E1 6501.523,E2 6501.523} C_VEL
LIN {X 0,Y 155.058,Z 1145.435,A -85,B 0,C 180,E1 6494.705,E2 6494.705} C_VEL
LIN {X 0,Y 173.612,Z 1138.948,A -85,B 0,C 180,E1 6489.996,E2 6489.996} C_VEL
LIN {X 0,Y 195.941,Z 1130.012,A -85,B 0,C 180,E1 6485.699,E2 6485.699} C_VEL
LIN {X 0,Y 219.14,Z 1119.022,A -85,B 0,C 180,E1 6482.261,E2 6482.261} C_VEL
LIN {X 0,Y 238.051,Z 1108.928,A -85,B 0,C 180,E1 6480,E2 6480} C_VEL
LIN {X 0,Y 254.069,Z 1099.454,A -85,B 0,C 180,E1 6478.358,E2 6478.358} C_VEL
LIN {X 0,Y 234.416,Z 1111.886,A -85,B 0,C 180,E1 6476.455,E2 6476.455} C_VEL
LIN {X 0,Y 212.766,Z 1124.284,A -85,B 0,C 180,E1 6473.882,E2 6473.882} C_VEL
LIN {X 0,Y 206.165,Z 1127.719,A -85,B 0,C 180,E1 6473.276,E2 6473.276} C_VEL
LIN {X 0,Y 186.946,Z 1136.293,A -85,B 0,C 180,E1 6472.421,E2 6472.421} C_VEL
LIN {X 0,Y 181.207,Z 1138.818,A -85,B 0,C 180,E1 6471.732,E2 6471.732} C_VEL
LIN {X 0,Y 155.309,Z 1149.621,A -85,B 0,C 180,E1 6466.439,E2 6466.439} C_VEL
LIN {X 0,Y 135.052,Z 1157.004,A -85,B 0,C 180,E1 6460.539,E2 6460.539} C_VEL
LIN {X 0,Y 117.402,Z 1162.803,A -85,B 0,C 180,E1 6453.167,E2 6453.167} C_VEL
LIN {X 0,Y 99.696,Z 1168.182,A -85,B 0,C 180,E1 6441.469,E2 6441.469} C_VEL
LIN {X 0,Y 87.414,Z 1171.602,A -85,B 0,C 180,E1 6426.498,E2 6426.498} C_VEL
LIN {X 0,Y 82.098,Z 1173.249,A -85,B 0,C 180,E1 6412.182,E2 6412.182} C_VEL
LIN {X 0,Y 80.899,Z 1173.799,A -85,B 0,C 180,E1 6399.246,E2 6399.246} C_VEL
LIN {X 0,Y 81.184,Z 1173.699,A -85,B 0,C 180,E1 6390.706,E2 6390.706} C_VEL
LIN {X 0,Y 80.998,Z 1173.014,A -85,B 0,C 180,E1 6382.91,E2 6382.91} C_VEL
LIN {X 0,Y 81.655,Z 1171.324,A -85,B 0,C 180,E1 6370.695,E2 6370.695} C_VEL
LIN {X 0,Y 85.789,Z 1168.284,A -85,B 0,C 180,E1 6356.786,E2 6356.786} C_VEL
LIN {X 0,Y 93.759,Z 1164.153,A -85,B 0,C 180,E1 6344.399,E2 6344.399} C_VEL
LIN {X 0,Y 105.646,Z 1158.637,A -85,B 0,C 180,E1 6333.608,E2 6333.608} C_VEL
LIN {X 0,Y 123.321,Z 1150.513,A -85,B 0,C 180,E1 6323.627,E2 6323.627} C_VEL
LIN {X 0,Y 142.795,Z 1140.779,A -85,B 0,C 180,E1 6316.408,E2 6316.408} C_VEL
LIN {X 0,Y 160.309,Z 1131.351,A -85,B 0,C 180,E1 6311.703,E2 6311.703} C_VEL
LIN {X 0,Y 180.546,Z 1119.488,A -85,B 0,C 180,E1 6307.566,E2 6307.566} C_VEL
LIN {X 0,Y 202.491,Z 1105.041,A -85,B 0,C 180,E1 6304.109,E2 6304.109} C_VEL
LIN {X 0,Y 220.578,Z 1091.869,A -85,B 0,C 180,E1 6301.818,E2 6301.818} C_VEL
LIN {X 0,Y 237.965,Z 1077.993,A -85,B 0,C 180,E1 6299.966,E2 6299.966} C_VEL
LIN {X 0,Y 259.108,Z 1059.265,A -85,B 0,C 180,E1 6298.08,E2 6298.08} C_VEL
LIN {X 0,Y 277,Z 1041.385,A -85,B 0,C 180,E1 6296.723,E2 6296.723} C_VEL
LIN {X 0,Y 291.762,Z 1025.14,A -85,B 0,C 180,E1 6295.745,E2 6295.745} C_VEL
LIN {X 0,Y 308.749,Z 1004.478,A -85,B 0,C 180,E1 6294.753,E2 6294.753} C_VEL
LIN {X 0,Y 324.786,Z 982.12,A -85,B 0,C 180,E1 6293.91,E2 6293.91} C_VEL
LIN {X 0,Y 336.723,Z 963.51,A -85,B 0,C 180,E1 6293.35,E2 6293.35} C_VEL
LIN {X 0,Y 338.742,Z 960.195,A -85,B 0,C 180,E1 6293.261,E2 6293.261} C_VEL
LIN {X 0,Y 326.185,Z 979.661,A -85,B 0,C 180,E1 6292.579,E2 6292.579} C_VEL
LIN {X 0,Y 312.665,Z 998.411,A -85,B 0,C 180,E1 6291.783,E2 6291.783} C_VEL
LIN {X 0,Y 294.804,Z 1020.322,A -85,B 0,C 180,E1 6290.63,E2 6290.63} C_VEL
LIN {X 0,Y 279.606,Z 1036.821,A -85,B 0,C 180,E1 6289.541,E2 6289.541} C_VEL
LIN {X 0,Y 264.423,Z 1051.763,A -85,B 0,C 180,E1 6288.335,E2 6288.335} C_VEL
LIN {X 0,Y 247.489,Z 1066.887,A -85,B 0,C 180,E1 6286.815,E2 6286.815} C_VEL
LIN {X 0,Y 225.203,Z 1084.555,A -85,B 0,C 180,E1 6284.458,E2 6284.458} C_VEL
LIN {X 0,Y 206.941,Z 1097.405,A -85,B 0,C 180,E1 6282.142,E2 6282.142} C_VEL
LIN {X 0,Y 188.166,Z 1109.344,A -85,B 0,C 180,E1 6279.261,E2 6279.261} C_VEL
LIN {X 0,Y 165.651,Z 1122.028,A -85,B 0,C 180,E1 6274.875,E2 6274.875} C_VEL
LIN {X 0,Y 147.462,Z 1131.121,A -85,B 0,C 180,E1 6270.215,E2 6270.215} C_VEL
LIN {X 0,Y 130.04,Z 1139.043,A -85,B 0,C 180,E1 6264.241,E2 6264.241} C_VEL
LIN {X 0,Y 110.286,Z 1147.178,A -85,B 0,C 180,E1 6254.255,E2 6254.255} C_VEL
LIN {X 0,Y 97.737,Z 1152.032,A -85,B 0,C 180,E1 6244.239,E2 6244.239} C_VEL
LIN {X 0,Y 88.73,Z 1155.625,A -85,B 0,C 180,E1 6232.527,E2 6232.527} C_VEL
LIN {X 0,Y 83.429,Z 1158.136,A -85,B 0,C 180,E1 6219.658,E2 6219.658} C_VEL
LIN {X 0,Y 81.529,Z 1159.604,A -85,B 0,C 180,E1 6207.891,E2 6207.891} C_VEL
LIN {X 0,Y 81.414,Z 1160.471,A -85,B 0,C 180,E1 6197.228,E2 6197.228} C_VEL
LIN {X 0,Y 83.176,Z 1160.932,A -85,B 0,C 180,E1 6184.357,E2 6184.357} C_VEL
LIN {X 0,Y 89.187,Z 1160.52,A -85,B 0,C 180,E1 6169.673,E2 6169.673} C_VEL
LIN {X 0,Y 99.307,Z 1159.068,A -85,B 0,C 180,E1 6157.306,E2 6157.306} C_VEL
LIN {X 0,Y 114.213,Z 1156.259,A -85,B 0,C 180,E1 6146.518,E2 6146.518} C_VEL
LIN {X 0,Y 134.986,Z 1151.236,A -85,B 0,C 180,E1 6137.153,E2 6137.153} C_VEL
LIN {X 0,Y 153.995,Z 1145.655,A -85,B 0,C 180,E1 6131.357,E2 6131.357} C_VEL
LIN {X 0,Y 173.474,Z 1139.01,A -85,B 0,C 180,E1 6126.952,E2 6126.952} C_VEL
LIN {X 0,Y 198.202,Z 1129.119,A -85,B 0,C 180,E1 6122.756,E2 6122.756} C_VEL
LIN {X 0,Y 219.18,Z 1119.3,A -85,B 0,C 180,E1 6120,E2 6120} C_VEL
LIN {X 0,Y 233.269,Z 1112.005,A -85,B 0,C 180,E1 6118.446,E2 6118.446} C_VEL
LIN {X 0,Y 206.612,Z 1126.654,A -85,B 0,C 180,E1 6115.487,E2 6115.487} C_VEL
LIN {X 0,Y 185.577,Z 1136.817,A -85,B 0,C 180,E1 6112.465,E2 6112.465} C_VEL
LIN {X 0,Y 181.207,Z 1138.818,A -85,B 0,C 180,E1 6111.732,E2 6111.732} C_VEL
LIN {X 0,Y 174.459,Z 1141.699,A -85,B 0,C 180,E1 6110.901,E2 6110.901} C_VEL
LIN {X 0,Y 154.826,Z 1148.767,A -85,B 0,C 180,E1 6109.484,E2 6109.484} C_VEL
LIN {X 0,Y 149.044,Z 1150.738,A -85,B 0,C 180,E1 6108.502,E2 6108.502} C_VEL
LIN {X 0,Y 128.739,Z 1157.695,A -85,B 0,C 180,E1 6102.802,E2 6102.802} C_VEL
LIN {X 0,Y 104.93,Z 1164.761,A -85,B 0,C 180,E1 6092.398,E2 6092.398} C_VEL
LIN {X 0,Y 89.832,Z 1168.71,A -85,B 0,C 180,E1 6081.181,E2 6081.181} C_VEL
LIN {X 0,Y 79.46,Z 1171.3,A -85,B 0,C 180,E1 6067.555,E2 6067.555} C_VEL
LIN {X 0,Y 74.039,Z 1172.729,A -85,B 0,C 180,E1 6052.218,E2 6052.218} C_VEL
LIN {X 0,Y 72.936,Z 1173.111,A -85,B 0,C 180,E1 6038.674,E2 6038.674} C_VEL
LIN {X 0,Y 73.226,Z 1173.01,A -85,B 0,C 180,E1 6030.001,E2 6030.001} C_VEL
LIN {X 0,Y 72.978,Z 1172.154,A -85,B 0,C 180,E1 6020.538,E2 6020.538} C_VEL
LIN {X 0,Y 74.261,Z 1170.315,A -85,B 0,C 180,E1 6007.018,E2 6007.018} C_VEL
LIN {X 0,Y 79.505,Z 1167.221,A -85,B 0,C 180,E1 5992.403,E2 5992.403} C_VEL
LIN {X 0,Y 89.185,Z 1162.86,A -85,B 0,C 180,E1 5979.326,E2 5979.326} C_VEL
LIN {X 0,Y 105.468,Z 1156.038,A -85,B 0,C 180,E1 5966.985,E2 5966.985} C_VEL
LIN {X 0,Y 125.099,Z 1147.223,A -85,B 0,C 180,E1 5957.991,E2 5957.991} C_VEL
LIN {X 0,Y 142.39,Z 1138.896,A -85,B 0,C 180,E1 5952.565,E2 5952.565} C_VEL
LIN {X 0,Y 161.586,Z 1128.819,A -85,B 0,C 180,E1 5948.095,E2 5948.095} C_VEL
LIN {X 0,Y 185.413,Z 1114.766,A -85,B 0,C 180,E1 5943.951,E2 5943.951} C_VEL
LIN {X 0,Y 204.296,Z 1102.32,A -85,B 0,C 180,E1 5941.402,E2 5941.402} C_VEL
LIN {X 0,Y 221.978,Z 1089.516,A -85,B 0,C 180,E1 5939.435,E2 5939.435} C_VEL
LIN {X 0,Y 243.2,Z 1072.507,A -85,B 0,C 180,E1 5937.476,E2 5937.476} C_VEL
LIN {X 0,Y 262.096,Z 1055.373,A -85,B 0,C 180,E1 5936.012,E2 5936.012} C_VEL
LIN {X 0,Y 278.043,Z 1039.438,A -85,B 0,C 180,E1 5934.939,E2 5934.939} C_VEL
LIN {X 0,Y 295.056,Z 1020.668,A -85,B 0,C 180,E1 5933.94,E2 5933.94} C_VEL
LIN {X 0,Y 310.483,Z 1001.6,A -85,B 0,C 180,E1 5933.145,E2 5933.145} C_VEL
LIN {X 0,Y 292.742,Z 1022.767,A -85,B 0,C 180,E1 5932.091,E2 5932.091} C_VEL
LIN {X 0,Y 277.322,Z 1039.186,A -85,B 0,C 180,E1 5931.07,E2 5931.07} C_VEL
LIN {X 0,Y 260.611,Z 1055.261,A -85,B 0,C 180,E1 5929.835,E2 5929.835} C_VEL
LIN {X 0,Y 239.188,Z 1073.541,A -85,B 0,C 180,E1 5928.006,E2 5928.006} C_VEL
LIN {X 0,Y 221.342,Z 1087.054,A -85,B 0,C 180,E1 5926.217,E2 5926.217} C_VEL
LIN {X 0,Y 203.727,Z 1099.12,A -85,B 0,C 180,E1 5924.139,E2 5924.139} C_VEL
LIN {X 0,Y 181.904,Z 1112.542,A -85,B 0,C 180,E1 5920.982,E2 5920.982} C_VEL
LIN {X 0,Y 160.691,Z 1123.874,A -85,B 0,C 180,E1 5917.056,E2 5917.056} C_VEL
LIN {X 0,Y 142.839,Z 1132.441,A -85,B 0,C 180,E1 5912.746,E2 5912.746} C_VEL
LIN {X 0,Y 122.05,Z 1141.439,A -85,B 0,C 180,E1 5905.833,E2 5905.833} C_VEL
LIN {X 0,Y 103.405,Z 1148.477,A -85,B 0,C 180,E1 5896.485,E2 5896.485} C_VEL
LIN {X 0,Y 90.18,Z 1153.214,A -85,B 0,C 180,E1 5885.988,E2 5885.988} C_VEL
LIN {X 0,Y 79.969,Z 1156.988,A -85,B 0,C 180,E1 5872.029,E2 5872.029} C_VEL
LIN {X 0,Y 74.319,Z 1159.706,A -85,B 0,C 180,E1 5854.63,E2 5854.63} C_VEL
LIN {X 0,Y 73.353,Z 1160.884,A -85,B 0,C 180,E1 5841.376,E2 5841.376} C_VEL
LIN {X 0,Y 74.396,Z 1161.513,A -85,B 0,C 180,E1 5827.894,E2 5827.894} C_VEL
LIN {X 0,Y 80.566,Z 1161.442,A -85,B 0,C 180,E1 5809.808,E2 5809.808} C_VEL
LIN {X 0,Y 92.545,Z 1159.967,A -85,B 0,C 180,E1 5794.804,E2 5794.804} C_VEL
LIN {X 0,Y 106.724,Z 1157.573,A -85,B 0,C 180,E1 5784.665,E2 5784.665} C_VEL
LIN {X 0,Y 125.836,Z 1153.52,A -85,B 0,C 180,E1 5775.964,E2 5775.964} C_VEL
LIN {X 0,Y 148.841,Z 1147.292,A -85,B 0,C 180,E1 5769.071,E2 5769.071} C_VEL
LIN {X 0,Y 169.16,Z 1140.697,A -85,B 0,C 180,E1 5764.747,E2 5764.747} C_VEL
LIN {X 0,Y 190.027,Z 1132.844,A -85,B 0,C 180,E1 5761.363,E2 5761.363} C_VEL
LIN {X 0,Y 212.39,Z 1123.114,A -85,B 0,C 180,E1 5758.529,E2 5758.529} C_VEL
LIN {X 0,Y 186.858,Z 1135.393,A -85,B 0,C 180,E1 5755.396,E2 5755.396} C_VEL
LIN {X 0,Y 166.021,Z 1144.256,A -85,B 0,C 180,E1 5752.038,E2 5752.038} C_VEL
LIN {X 0,Y 149.044,Z 1150.738,A -85,B 0,C 180,E1 5748.502,E2 5748.502} C_VEL
LIN {X 0,Y 142.279,Z 1153.093,A -85,B 0,C 180,E1 5747.295,E2 5747.295} C_VEL
LIN {X 0,Y 122.029,Z 1158.652,A -85,B 0,C 180,E1 5744.744,E2 5744.744} C_VEL
LIN {X 0,Y 116.846,Z 1159.97,A -85,B 0,C 180,E1 5743.342,E2 5743.342} C_VEL
LIN {X 0,Y 98.202,Z 1164.922,A -85,B 0,C 180,E1 5734.982,E2 5734.982} C_VEL
LIN {X 0,Y 82.316,Z 1168.661,A -85,B 0,C 180,E1 5723.291,E2 5723.291} C_VEL
LIN {X 0,Y 69.369,Z 1171.519,A -85,B 0,C 180,E1 5704.204,E2 5704.204} C_VEL
LIN {X 0,Y 65.066,Z 1172.438,A -85,B 0,C 180,E1 5684.5,E2 5684.5} C_VEL
LIN {X 0,Y 65.17,Z 1172.383,A -85,B 0,C 180,E1 5672.639,E2 5672.639} C_VEL
LIN {X 0,Y 65.134,Z 1171.979,A -85,B 0,C 180,E1 5665.599,E2 5665.599} C_VEL
LIN {X 0,Y 65.625,Z 1170.481,A -85,B 0,C 180,E1 5650.416,E2 5650.416} C_VEL
LIN {X 0,Y 71.217,Z 1167.256,A -85,B 0,C 180,E1 5631.836,E2 5631.836} C_VEL
LIN {X 0,Y 81.647,Z 1162.965,A -85,B 0,C 180,E1 5617.251,E2 5617.251} C_VEL
LIN {X 0,Y 95.055,Z 1157.754,A -85,B 0,C 180,E1 5606.609,E2 5606.609} C_VEL
LIN {X 0,Y 113.275,Z 1150.409,A -85,B 0,C 180,E1 5597.581,E2 5597.581} C_VEL
LIN {X 0,Y 136.173,Z 1140.127,A -85,B 0,C 180,E1 5590.297,E2 5590.297} C_VEL
LIN {X 0,Y 154.861,Z 1130.787,A -85,B 0,C 180,E1 5586.124,E2 5586.124} C_VEL
LIN {X 0,Y 173.207,Z 1120.688,A -85,B 0,C 180,E1 5582.97,E2 5582.97} C_VEL
LIN {X 0,Y 195.971,Z 1106.799,A -85,B 0,C 180,E1 5579.927,E2 5579.927} C_VEL
LIN {X 0,Y 217.775,Z 1091.571,A -85,B 0,C 180,E1 5577.632,E2 5577.632} C_VEL
LIN {X 0,Y 235.514,Z 1077.877,A -85,B 0,C 180,E1 5576.089,E2 5576.089} C_VEL
LIN {X 0,Y 256.621,Z 1059.849,A -85,B 0,C 180,E1 5574.553,E2 5574.553} C_VEL
LIN {X 0,Y 276.189,Z 1040.765,A -85,B 0,C 180,E1 5573.347,E2 5573.347} C_VEL
LIN {X 0,Y 281.752,Z 1035.007,A -85,B 0,C 180,E1 5573.029,E2 5573.029} C_VEL
LIN {X 0,Y 264.586,Z 1051.745,A -85,B 0,C 180,E1 5571.924,E2 5571.924} C_VEL
LIN {X 0,Y 248.128,Z 1066.241,A -85,B 0,C 180,E1 5570.724,E2 5570.724} C_VEL
LIN {X 0,Y 227.18,Z 1082.846,A -85,B 0,C 180,E1 5568.948,E2 5568.948} C_VEL
LIN {X 0,Y 206.222,Z 1097.304,A -85,B 0,C 180,E1 5566.827,E2 5566.827} C_VEL
LIN {X 0,Y 187.697,Z 1108.773,A -85,B 0,C 180,E1 5564.552,E2 5564.552} C_VEL
LIN {X 0,Y 165.831,Z 1120.895,A -85,B 0,C 180,E1 5561.192,E2 5561.192} C_VEL
LIN {X 0,Y 143.686,Z 1131.466,A -85,B 0,C 180,E1 5556.713,E2 5556.713} C_VEL
LIN {X 0,Y 125.056,Z 1139.364,A -85,B 0,C 180,E1 5551.579,E2 5551.579} C_VEL
LIN {X 0,Y 105.359,Z 1146.856,A -85,B 0,C 180,E1 5543.769,E2 5543.769} C_VEL
LIN {X 0,Y 86.842,Z 1153.05,A -85,B 0,C 180,E1 5531.896,E2 5531.896} C_VEL
LIN {X 0,Y 75.132,Z 1156.857,A -85,B 0,C 180,E1 5518.625,E2 5518.625} C_VEL
LIN {X 0,Y 68.23,Z 1159.389,A -85,B 0,C 180,E1 5503.56,E2 5503.56} C_VEL
LIN {X 0,Y 65.646,Z 1160.879,A -85,B 0,C 180,E1 5489.127,E2 5489.127} C_VEL
LIN {X 0,Y 65.475,Z 1161.744,A -85,B 0,C 180,E1 5476.757,E2 5476.757} C_VEL
LIN {X 0,Y 68.056,Z 1162.282,A -85,B 0,C 180,E1 5460.031,E2 5460.031} C_VEL
LIN {X 0,Y 76.224,Z 1161.9,A -85,B 0,C 180,E1 5442.728,E2 5442.728} C_VEL
LIN {X 0,Y 88.634,Z 1160.499,A -85,B 0,C 180,E1 5429.701,E2 5429.701} C_VEL
LIN {X 0,Y 105.378,Z 1157.837,A -85,B 0,C 180,E1 5419.396,E2 5419.396} C_VEL
LIN {X 0,Y 130.04,Z 1152.539,A -85,B 0,C 180,E1 5410.207,E2 5410.207} C_VEL
LIN {X 0,Y 150.591,Z 1146.95,A -85,B 0,C 180,E1 5405.165,E2 5405.165} C_VEL
LIN {X 0,Y 171.845,Z 1140.099,A -85,B 0,C 180,E1 5401.334,E2 5401.334} C_VEL
LIN {X 0,Y 191.387,Z 1132.765,A -85,B 0,C 180,E1 5398.608,E2 5398.608} C_VEL
LIN {X 0,Y 168.495,Z 1142.434,A -85,B 0,C 180,E1 5395.505,E2 5395.505} C_VEL
LIN {X 0,Y 147.515,Z 1150.253,A -85,B 0,C 180,E1 5391.725,E2 5391.725} C_VEL
LIN {X 0,Y 123.835,Z 1158.002,A -85,B 0,C 180,E1 5385.672,E2 5385.672} C_VEL
LIN {X 0,Y 116.846,Z 1159.97,A -85,B 0,C 180,E1 5383.342,E2 5383.342} C_VEL
LIN {X 0,Y 110.245,Z 1161.661,A -85,B 0,C 180,E1 5381.452,E2 5381.452} C_VEL
LIN {X 0,Y 90.438,Z 1165.543,A -85,B 0,C 180,E1 5376.702,E2 5376.702} C_VEL
LIN {X 0,Y 85.619,Z 1166.435,A -85,B 0,C 180,E1 5374.322,E2 5374.322} C_VEL
LIN {X 0,Y 69.342,Z 1169.589,A -85,B 0,C 180,E1 5359.542,E2 5359.542} C_VEL
LIN {X 0,Y 60.228,Z 1171.202,A -85,B 0,C 180,E1 5342.09,E2 5342.09} C_VEL
LIN {X 0,Y 57.069,Z 1171.752,A -85,B 0,C 180,E1 5324.199,E2 5324.199} C_VEL
LIN {X 0,Y 57.25,Z 1171.678,A -85,B 0,C 180,E1 5311.001,E2 5311.001} C_VEL
LIN {X 0,Y 57.038,Z 1171.049,A -85,B 0,C 180,E1 5301.939,E2 5301.939} C_VEL
LIN {X 0,Y 58.443,Z 1169.389,A -85,B 0,C 180,E1 5285.063,E2 5285.063} C_VEL
LIN {X 0,Y 64.861,Z 1166.465,A -85,B 0,C 180,E1 5267.291,E2 5267.291} C_VEL
LIN {X 0,Y 76.175,Z 1162.366,A -85,B 0,C 180,E1 5252.856,E2 5252.856} C_VEL
LIN {X 0,Y 90.777,Z 1157.167,A -85,B 0,C 180,E1 5242.301,E2 5242.301} C_VEL
LIN {X 0,Y 109.229,Z 1150.173,A -85,B 0,C 180,E1 5234,E2 5234} C_VEL
LIN {X 0,Y 133.013,Z 1140.023,A -85,B 0,C 180,E1 5227.143,E2 5227.143} C_VEL
LIN {X 0,Y 153.204,Z 1130.255,A -85,B 0,C 180,E1 5223.117,E2 5223.117} C_VEL
LIN {X 0,Y 171.976,Z 1120.168,A -85,B 0,C 180,E1 5220.261,E2 5220.261} C_VEL
LIN {X 0,Y 195.154,Z 1106.293,A -85,B 0,C 180,E1 5217.522,E2 5217.522} C_VEL
LIN {X 0,Y 216.813,Z 1091.418,A -85,B 0,C 180,E1 5215.503,E2 5215.503} C_VEL
LIN {X 0,Y 235.217,Z 1077.405,A -85,B 0,C 180,E1 5214.089,E2 5214.089} C_VEL
LIN {X 0,Y 252.885,Z 1062.561,A -85,B 0,C 180,E1 5212.931,E2 5212.931} C_VEL
LIN {X 0,Y 235.439,Z 1076.682,A -85,B 0,C 180,E1 5211.688,E2 5211.688} C_VEL
LIN {X 0,Y 218.109,Z 1089.357,A -85,B 0,C 180,E1 5210.265,E2 5210.265} C_VEL
LIN {X 0,Y 198.076,Z 1102.542,A -85,B 0,C 180,E1 5208.316,E2 5208.316} C_VEL
LIN {X 0,Y 174.557,Z 1116.046,A -85,B 0,C 180,E1 5205.471,E2 5205.471} C_VEL
LIN {X 0,Y 155.178,Z 1125.827,A -85,B 0,C 180,E1 5202.479,E2 5202.479} C_VEL
LIN {X 0,Y 135.395,Z 1134.7,A -85,B 0,C 180,E1 5198.509,E2 5198.509} C_VEL
LIN {X 0,Y 110.806,Z 1144.214,A -85,B 0,C 180,E1 5191.428,E2 5191.428} C_VEL
LIN {X 0,Y 93.145,Z 1150.137,A -85,B 0,C 180,E1 5183.617,E2 5183.617} C_VEL
LIN {X 0,Y 77.848,Z 1154.807,A -85,B 0,C 180,E1 5172.899,E2 5172.899} C_VEL
LIN {X 0,Y 64.237,Z 1158.949,A -85,B 0,C 180,E1 5154.85,E2 5154.85} C_VEL
LIN {X 0,Y 58.121,Z 1161.254,A -85,B 0,C 180,E1 5133.784,E2 5133.784} C_VEL
LIN {X 0,Y 57.422,Z 1162.296,A -85,B 0,C 180,E1 5118.957,E2 5118.957} C_VEL
LIN {X 0,Y 59.636,Z 1162.948,A -85,B 0,C 180,E1 5100.907,E2 5100.907} C_VEL
LIN {X 0,Y 69.638,Z 1162.642,A -85,B 0,C 180,E1 5079.164,E2 5079.164} C_VEL
LIN {X 0,Y 83.99,Z 1161.214,A -85,B 0,C 180,E1 5065.211,E2 5065.211} C_VEL
LIN {X 0,Y 101.637,Z 1158.627,A -85,B 0,C 180,E1 5055.403,E2 5055.403} C_VEL
LIN {X 0,Y 125.969,Z 1153.778,A -85,B 0,C 180,E1 5047.173,E2 5047.173} C_VEL
LIN {X 0,Y 148.094,Z 1148.028,A -85,B 0,C 180,E1 5042.256,E2 5042.256} C_VEL
LIN {X 0,Y 169.01,Z 1141.524,A -85,B 0,C 180,E1 5038.864,E2 5038.864} C_VEL
LIN {X 0,Y 170.257,Z 1141.11,A -85,B 0,C 180,E1 5038.691,E2 5038.691} C_VEL
LIN {X 0,Y 148.466,Z 1149.088,A -85,B 0,C 180,E1 5035.36,E2 5035.36} C_VEL
LIN {X 0,Y 126.625,Z 1156.047,A -85,B 0,C 180,E1 5030.762,E2 5030.762} C_VEL
LIN {X 0,Y 100.758,Z 1162.997,A -85,B 0,C 180,E1 5022.298,E2 5022.298} C_VEL
LIN {X 0,Y 85.619,Z 1166.435,A -85,B 0,C 180,E1 5014.322,E2 5014.322} C_VEL
LIN {X 0,Y 79.581,Z 1167.473,A -85,B 0,C 180,E1 5011.002,E2 5011.002} C_VEL
LIN {X 0,Y 61.617,Z 1169.503,A -85,B 0,C 180,E1 5000.966,E2 5000.966} C_VEL
LIN {X 0,Y 57.866,Z 1170.001,A -85,B 0,C 180,E1 4996.349,E2 4996.349} C_VEL
LIN {X 0,Y 49.542,Z 1171.063,A -85,B 0,C 180,E1 4970.066,E2 4970.066} C_VEL
LIN {X 0,Y 49.225,Z 1171.025,A -85,B 0,C 180,E1 4952.329,E2 4952.329} C_VEL
LIN {X 0,Y 49.119,Z 1170.569,A -85,B 0,C 180,E1 4944.159,E2 4944.159} C_VEL
LIN {X 0,Y 50.471,Z 1168.983,A -85,B 0,C 180,E1 4924.163,E2 4924.163} C_VEL
LIN {X 0,Y 58.463,Z 1165.854,A -85,B 0,C 180,E1 4902.659,E2 4902.659} C_VEL
LIN {X 0,Y 71.218,Z 1161.766,A -85,B 0,C 180,E1 4887.813,E2 4887.813} C_VEL
LIN {X 0,Y 87.059,Z 1156.581,A -85,B 0,C 180,E1 4877.592,E2 4877.592} C_VEL
LIN {X 0,Y 106.561,Z 1149.6,A -85,B 0,C 180,E1 4869.869,E2 4869.869} C_VEL
LIN {X 0,Y 132.221,Z 1139.034,A -85,B 0,C 180,E1 4863.454,E2 4863.454} C_VEL
LIN {X 0,Y 152.34,Z 1129.538,A -85,B 0,C 180,E1 4860,E2 4860} C_VEL
LIN {X 0,Y 172.642,Z 1118.811,A -85,B 0,C 180,E1 4857.344,E2 4857.344} C_VEL
LIN {X 0,Y 196.746,Z 1104.422,A -85,B 0,C 180,E1 4854.915,E2 4854.915} C_VEL
LIN {X 0,Y 217.47,Z 1090.309,A -85,B 0,C 180,E1 4853.263,E2 4853.263} C_VEL
LIN {X 0,Y 223.477,Z 1085.97,A -85,B 0,C 180,E1 4852.839,E2 4852.839} C_VEL
LIN {X 0,Y 203.965,Z 1099.017,A -85,B 0,C 180,E1 4851.259,E2 4851.259} C_VEL
LIN {X 0,Y 184.766,Z 1110.505,A -85,B 0,C 180,E1 4849.397,E2 4849.397} C_VEL
LIN {X 0,Y 161.404,Z 1122.882,A -85,B 0,C 180,E1 4846.55,E2 4846.55} C_VEL
LIN {X 0,Y 139.081,Z 1132.956,A -85,B 0,C 180,E1 4842.966,E2 4842.966} C_VEL
LIN {X 0,Y 120.076,Z 1140.497,A -85,B 0,C 180,E1 4838.844,E2 4838.844} C_VEL
LIN {X 0,Y 99.294,Z 1147.733,A -85,B 0,C 180,E1 4832.39,E2 4832.39} C_VEL
LIN {X 0,Y 77.908,Z 1154.062,A -85,B 0,C 180,E1 4821.523,E2 4821.523} C_VEL
LIN {X 0,Y 63.313,Z 1157.938,A -85,B 0,C 180,E1 4808.017,E2 4808.017} C_VEL
LIN {X 0,Y 53.873,Z 1160.531,A -85,B 0,C 180,E1 4790.648,E2 4790.648} C_VEL
LIN {X 0,Y 49.919,Z 1162.082,A -85,B 0,C 180,E1 4772.295,E2 4772.295} C_VEL
LIN {X 0,Y 49.565,Z 1163.026,A -85,B 0,C 180,E1 4755.542,E2 4755.542} C_VEL
LIN {X 0,Y 53.179,Z 1163.635,A -85,B 0,C 180,E1 4734.348,E2 4734.348} C_VEL
LIN {X 0,Y 64.631,Z 1163.291,A -85,B 0,C 180,E1 4713.342,E2 4713.342} C_VEL
LIN {X 0,Y 79.919,Z 1161.929,A -85,B 0,C 180,E1 4700.228,E2 4700.228} C_VEL
LIN {X 0,Y 98.798,Z 1159.362,A -85,B 0,C 180,E1 4690.987,E2 4690.987} C_VEL
LIN {X 0,Y 124.213,Z 1154.553,A -85,B 0,C 180,E1 4683.487,E2 4683.487} C_VEL
LIN {X 0,Y 146.998,Z 1148.822,A -85,B 0,C 180,E1 4679.091,E2 4679.091} C_VEL
LIN {X 0,Y 148.736,Z 1148.345,A -85,B 0,C 180,E1 4678.748,E2 4678.748} C_VEL
LIN {X 0,Y 126.504,Z 1155.23,A -85,B 0,C 180,E1 4674.796,E2 4674.796} C_VEL
LIN {X 0,Y 99.41,Z 1162.21,A -85,B 0,C 180,E1 4667.322,E2 4667.322} C_VEL
LIN {X 0,Y 78.94,Z 1166.413,A -85,B 0,C 180,E1 4657.612,E2 4657.612} C_VEL
LIN {X 0,Y 63.108,Z 1169.115,A -85,B 0,C 180,E1 4643.905,E2 4643.905} C_VEL
LIN {X 0,Y 57.866,Z 1170.001,A -85,B 0,C 180,E1 4636.349,E2 4636.349} C_VEL
LIN {X 0,Y 53.512,Z 1170.484,A -85,B 0,C 180,E1 4629.756,E2 4629.756} C_VEL
LIN {X 0,Y 45.205,Z 1170.605,A -85,B 0,C 180,E1 4616.582,E2 4616.582} C_VEL
LIN {X 0,Y 41.208,Z 1170.394,A -85,B 0,C 180,E1 4602.582,E2 4602.582} C_VEL
LIN {X 0,Y 41.046,Z 1170.374,A -85,B 0,C 180,E1 4598.675,E2 4598.675} C_VEL
LIN {X 0,Y 41.289,Z 1170.154,A -85,B 0,C 180,E1 4588.613,E2 4588.613} C_VEL
LIN {X 0,Y 41.812,Z 1168.982,A -85,B 0,C 180,E1 4567.505,E2 4567.505} C_VEL
LIN {X 0,Y 51.329,Z 1165.61,A -85,B 0,C 180,E1 4538.815,E2 4538.815} C_VEL
LIN {X 0,Y 66.094,Z 1161.401,A -85,B 0,C 180,E1 4522.663,E2 4522.663} C_VEL
LIN {X 0,Y 83.977,Z 1155.994,A -85,B 0,C 180,E1 4512.495,E2 4512.495} C_VEL
LIN {X 0,Y 103.516,Z 1149.364,A -85,B 0,C 180,E1 4505.807,E2 4505.807} C_VEL
LIN {X 0,Y 128.982,Z 1139.37,A -85,B 0,C 180,E1 4500.246,E2 4500.246} C_VEL
LIN {X 0,Y 151.192,Z 1129.178,A -85,B 0,C 180,E1 4496.949,E2 4496.949} C_VEL
LIN {X 0,Y 171.722,Z 1118.552,A -85,B 0,C 180,E1 4494.653,E2 4494.653} C_VEL
LIN {X 0,Y 193.533,Z 1105.885,A -85,B 0,C 180,E1 4492.716,E2 4492.716} C_VEL
LIN {X 0,Y 171.26,Z 1118.064,A -85,B 0,C 180,E1 4490.631,E2 4490.631} C_VEL
LIN {X 0,Y 151.148,Z 1127.769,A -85,B 0,C 180,E1 4488.245,E2 4488.245} C_VEL
LIN {X 0,Y 127.608,Z 1137.716,A -85,B 0,C 180,E1 4484.524,E2 4484.524} C_VEL
LIN {X 0,Y 103.831,Z 1146.033,A -85,B 0,C 180,E1 4479.078,E2 4479.078} C_VEL
LIN {X 0,Y 84.665,Z 1151.795,A -85,B 0,C 180,E1 4472.339,E2 4472.339} C_VEL
LIN {X 0,Y 65.573,Z 1156.785,A -85,B 0,C 180,E1 4461.045,E2 4461.045} C_VEL
LIN {X 0,Y 48.73,Z 1160.729,A -85,B 0,C 180,E1 4439.5,E2 4439.5} C_VEL
LIN {X 0,Y 42.216,Z 1162.649,A -85,B 0,C 180,E1 4415.435,E2 4415.435} C_VEL
LIN {X 0,Y 41.55,Z 1163.632,A -85,B 0,C 180,E1 4396.075,E2 4396.075} C_VEL
LIN {X 0,Y 45.439,Z 1164.306,A -85,B 0,C 180,E1 4371.965,E2 4371.965} C_VEL
LIN {X 0,Y 59.666,Z 1163.988,A -85,B 0,C 180,E1 4347.356,E2 4347.356} C_VEL
LIN {X 0,Y 77.384,Z 1162.556,A -85,B 0,C 180,E1 4334.289,E2 4334.289} C_VEL
LIN {X 0,Y 98.116,Z 1159.879,A -85,B 0,C 180,E1 4325.849,E2 4325.849} C_VEL
LIN {X 0,Y 125.997,Z 1154.628,A -85,B 0,C 180,E1 4319.134,E2 4319.134} C_VEL
LIN {X 0,Y 127.35,Z 1154.315,A -85,B 0,C 180,E1 4318.885,E2 4318.885} C_VEL
LIN {X 0,Y 100.738,Z 1161.045,A -85,B 0,C 180,E1 4312.998,E2 4312.998} C_VEL
LIN {X 0,Y 76.992,Z 1165.646,A -85,B 0,C 180,E1 4303.946,E2 4303.946} C_VEL
LIN {X 0,Y 59.291,Z 1168.371,A -85,B 0,C 180,E1 4291.273,E2 4291.273} C_VEL
LIN {X 0,Y 47.03,Z 1169.865,A -85,B 0,C 180,E1 4272.87,E2 4272.87} C_VEL
LIN {X 0,Y 41.468,Z 1170.378,A -85,B 0,C 180,E1 4249.729,E2 4249.729} C_VEL
LIN {X 0,Y 41.046,Z 1170.374,A -85,B 0,C 180,E1 4238.675,E2 4238.675} C_VEL
LIN {X 0,Y 40.53,Z 1170.223,A -85,B 0,C 180,E1 4231.051,E2 4231.051} C_VEL
LIN {X 0,Y 38.819,Z 1169.668,A -85,B 0,C 180,E1 4220.961,E2 4220.961} C_VEL
LIN {X 0,Y 37.112,Z 1167.352,A -85,B 0,C 180,E1 4191.235,E2 4191.235} C_VEL
LIN {X 0,Y 38.633,Z 1166.806,A -85,B 0,C 180,E1 4185.567,E2 4185.567} C_VEL
LIN {X 0,Y 51.734,Z 1163.53,A -85,B 0,C 180,E1 4164.723,E2 4164.723} C_VEL
LIN {X 0,Y 73.792,Z 1157.789,A -85,B 0,C 180,E1 4150.146,E2 4150.146} C_VEL
LIN {X 0,Y 97.075,Z 1150.472,A -85,B 0,C 180,E1 4142.459,E2 4142.459} C_VEL
LIN {X 0,Y 118.042,Z 1142.854,A -85,B 0,C 180,E1 4138.175,E2 4138.175} C_VEL
LIN {X 0,Y 142.583,Z 1132.592,A -85,B 0,C 180,E1 4134.726,E2 4134.726} C_VEL
LIN {X 0,Y 163.102,Z 1122.612,A -85,B 0,C 180,E1 4132.627,E2 4132.627} C_VEL
LIN {X 0,Y 138.155,Z 1133.667,A -85,B 0,C 180,E1 4129.819,E2 4129.819} C_VEL
LIN {X 0,Y 117.172,Z 1141.622,A -85,B 0,C 180,E1 4126.601,E2 4126.601} C_VEL
LIN {X 0,Y 95.728,Z 1148.601,A -85,B 0,C 180,E1 4121.892,E2 4121.892} C_VEL
LIN {X 0,Y 70.822,Z 1155.267,A -85,B 0,C 180,E1 4112.801,E2 4112.801} C_VEL
LIN {X 0,Y 52.424,Z 1159.315,A -85,B 0,C 180,E1 4099.719,E2 4099.719} C_VEL
LIN {X 0,Y 39.86,Z 1161.886,A -85,B 0,C 180,E1 4080.11,E2 4080.11} C_VEL
LIN {X 0,Y 34.095,Z 1163.419,A -85,B 0,C 180,E1 4055.046,E2 4055.046} C_VEL
LIN {X 0,Y 33.721,Z 1164.316,A -85,B 0,C 180,E1 4032.751,E2 4032.751} C_VEL
LIN {X 0,Y 39.96,Z 1164.984,A -85,B 0,C 180,E1 4002.501,E2 4002.501} C_VEL
LIN {X 0,Y 56.276,Z 1164.641,A -85,B 0,C 180,E1 3979.668,E2 3979.668} C_VEL
LIN {X 0,Y 74.796,Z 1163.275,A -85,B 0,C 180,E1 3968.417,E2 3968.417} C_VEL
LIN {X 0,Y 96.219,Z 1160.672,A -85,B 0,C 180,E1 3961.191,E2 3961.191} C_VEL
LIN {X 0,Y 105.431,Z 1159.247,A -85,B 0,C 180,E1 3958.988,E2 3958.988} C_VEL
LIN {X 0,Y 76.957,Z 1164.736,A -85,B 0,C 180,E1 3950.907,E2 3950.907} C_VEL
LIN {X 0,Y 56.572,Z 1167.626,A -85,B 0,C 180,E1 3939.51,E2 3939.51} C_VEL
LIN {X 0,Y 41.344,Z 1169.197,A -85,B 0,C 180,E1 3920.706,E2 3920.706} C_VEL
LIN {X 0,Y 33.701,Z 1169.693,A -85,B 0,C 180,E1 3892.688,E2 3892.688} C_VEL
LIN {X 0,Y 33.347,Z 1169.52,A -85,B 0,C 180,E1 3870.001,E2 3870.001} C_VEL
LIN {X 0,Y 33.923,Z 1168.429,A -85,B 0,C 180,E1 3845.631,E2 3845.631} C_VEL
LIN {X 0,Y 38.633,Z 1166.806,A -85,B 0,C 180,E1 3825.567,E2 3825.567} C_VEL
LIN {X 0,Y 42.015,Z 1165.766,A -85,B 0,C 180,E1 3815.741,E2 3815.741} C_VEL
LIN {X 0,Y 53.679,Z 1161.805,A -85,B 0,C 180,E1 3792.987,E2 3792.987} C_VEL
LIN {X 0,Y 58.124,Z 1160.603,A -85,B 0,C 180,E1 3789.746,E2 3789.746} C_VEL
LIN {X 0,Y 79.02,Z 1155.102,A -85,B 0,C 180,E1 3781.626,E2 3781.626} C_VEL
LIN {X 0,Y 100.135,Z 1148.543,A -85,B 0,C 180,E1 3776.859,E2 3776.859} C_VEL
LIN {X 0,Y 125.884,Z 1139.141,A -85,B 0,C 180,E1 3773.136,E2 3773.136} C_VEL
LIN {X 0,Y 131.359,Z 1136.802,A -85,B 0,C 180,E1 3772.483,E2 3772.483} C_VEL
LIN {X 0,Y 104.999,Z 1146.04,A -85,B 0,C 180,E1 3768.759,E2 3768.759} C_VEL
LIN {X 0,Y 82.087,Z 1152.539,A -85,B 0,C 180,E1 3763.73,E2 3763.73} C_VEL
LIN {X 0,Y 62.176,Z 1157.215,A -85,B 0,C 180,E1 3756.436,E2 3756.436} C_VEL
LIN {X 0,Y 42.156,Z 1161.119,A -85,B 0,C 180,E1 3741.507,E2 3741.507} C_VEL
LIN {X 0,Y 27.827,Z 1163.72,A -85,B 0,C 180,E1 3708.866,E2 3708.866} C_VEL
LIN {X 0,Y 25.509,Z 1164.708,A -85,B 0,C 180,E1 3678.505,E2 3678.505} C_VEL
LIN {X 0,Y 29.848,Z 1165.423,A -85,B 0,C 180,E1 3645.293,E2 3645.293} C_VEL
LIN {X 0,Y 46.939,Z 1165.635,A -85,B 0,C 180,E1 3616.552,E2 3616.552} C_VEL
LIN {X 0,Y 71.081,Z 1164.176,A -85,B 0,C 180,E1 3602.891,E2 3602.891} C_VEL
LIN {X 0,Y 82.999,Z 1163.087,A -85,B 0,C 180,E1 3599.113,E2 3599.113} C_VEL
LIN {X 0,Y 56.956,Z 1166.683,A -85,B 0,C 180,E1 3589.447,E2 3589.447} C_VEL
LIN {X 0,Y 38.146,Z 1168.424,A -85,B 0,C 180,E1 3573.025,E2 3573.025} C_VEL
LIN {X 0,Y 27.003,Z 1169,A -85,B 0,C 180,E1 3543.74,E2 3543.74} C_VEL
LIN {X 0,Y 25.356,Z 1168.818,A -85,B 0,C 180,E1 3510.002,E2 3510.002} C_VEL
LIN {X 0,Y 27.39,Z 1167.513,A -85,B 0,C 180,E1 3474.265,E2 3474.265} C_VEL
LIN {X 0,Y 42.062,Z 1164.206,A -85,B 0,C 180,E1 3442.02,E2 3442.02} C_VEL
LIN {X 0,Y 58.124,Z 1160.603,A -85,B 0,C 180,E1 3429.746,E2 3429.746} C_VEL
LIN {X 0,Y 64.389,Z 1158.926,A -85,B 0,C 180,E1 3425.775,E2 3425.775} C_VEL
LIN {X 0,Y 81.235,Z 1153.745,A -85,B 0,C 180,E1 3415.556,E2 3415.556} C_VEL
LIN {X 0,Y 86.75,Z 1152.133,A -85,B 0,C 180,E1 3414.091,E2 3414.091} C_VEL
LIN {X 0,Y 98.289,Z 1148.492,A -85,B 0,C 180,E1 3412.36,E2 3412.36} C_VEL
LIN {X 0,Y 77.511,Z 1154.034,A -85,B 0,C 180,E1 3408.623,E2 3408.623} C_VEL
LIN {X 0,Y 52.006,Z 1159.502,A -85,B 0,C 180,E1 3400.398,E2 3400.398} C_VEL
LIN {X 0,Y 30.307,Z 1162.921,A -85,B 0,C 180,E1 3382.351,E2 3382.351} C_VEL
LIN {X 0,Y 19.151,Z 1164.622,A -85,B 0,C 180,E1 3348.253,E2 3348.253} C_VEL
LIN {X 0,Y 17.772,Z 1165.492,A -85,B 0,C 180,E1 3310.27,E2 3310.27} C_VEL
LIN {X 0,Y 26.828,Z 1166.25,A -85,B 0,C 180,E1 3266.558,E2 3266.558} C_VEL
LIN {X 0,Y 50.283,Z 1166.077,A -85,B 0,C 180,E1 3243.42,E2 3243.42} C_VEL
LIN {X 0,Y 59.996,Z 1165.636,A -85,B 0,C 180,E1 3239.339,E2 3239.339} C_VEL
LIN {X 0,Y 36.956,Z 1167.648,A -85,B 0,C 180,E1 3226.911,E2 3226.911} C_VEL
LIN {X 0,Y 21.25,Z 1168.306,A -85,B 0,C 180,E1 3198.794,E2 3198.794} C_VEL
LIN {X 0,Y 17.347,Z 1168.115,A -85,B 0,C 180,E1 3150.002,E2 3150.002} C_VEL
LIN {X 0,Y 21.853,Z 1166.628,A -85,B 0,C 180,E1 3098.943,E2 3098.943} C_VEL
LIN {X 0,Y 39.69,Z 1163.41,A -85,B 0,C 180,E1 3070.745,E2 3070.745} C_VEL
LIN {X 0,Y 59.993,Z 1159.131,A -85,B 0,C 180,E1 3060.452,E2 3060.452} C_VEL
LIN {X 0,Y 81.326,Z 1153.641,A -85,B 0,C 180,E1 3055.063,E2 3055.063} C_VEL
LIN {X 0,Y 86.75,Z 1152.133,A -85,B 0,C 180,E1 3054.091,E2 3054.091} C_VEL
LIN {X 0,Y 85.353,Z 1152.427,A -85,B 0,C 180,E1 3053.408,E2 3053.408} C_VEL
LIN {X 0,Y 77.512,Z 1154.375,A -85,B 0,C 180,E1 3052.699,E2 3052.699} C_VEL
LIN {X 0,Y 59.872,Z 1158.608,A -85,B 0,C 180,E1 3053.119,E2 3053.119} C_VEL
LIN {X 0,Y 50.692,Z 1160.484,A -85,B 0,C 180,E1 3054.634,E2 3054.634} C_VEL
LIN {X 0,Y 26.155,Z 1164.676,A -85,B 0,C 180,E1 3066.586,E2 3066.586} C_VEL
LIN {X 0,Y 11.11,Z 1166.771,A -85,B 0,C 180,E1 3103.955,E2 3103.955} C_VEL
LIN {X 0,Y 9.281,Z 1167.408,A -85,B 0,C 180,E1 3150.004,E2 3150.004} C_VEL
LIN {X 0,Y 17,Z 1167.612,A -85,B 0,C 180,E1 3220.232,E2 3220.232} C_VEL
LIN {X 0,Y 35.444,Z 1167.003,A -85,B 0,C 180,E1 3239.715,E2 3239.715} C_VEL
LIN {X 0,Y 17.104,Z 1166.619,A -85,B 0,C 180,E1 3260.714,E2 3260.714} C_VEL
LIN {X 0,Y 9.548,Z 1165.895,A -85,B 0,C 180,E1 3317.907,E2 3317.907} C_VEL
LIN {X 0,Y 16.716,Z 1164.835,A -85,B 0,C 180,E1 3381.038,E2 3381.038} C_VEL
LIN {X 0,Y 38.357,Z 1162.044,A -85,B 0,C 180,E1 3404.679,E2 3404.679} C_VEL
LIN {X 0,Y 59.638,Z 1158.415,A -85,B 0,C 180,E1 3411.552,E2 3411.552} C_VEL
LIN {X 0,Y 61.954,Z 1157.966,A -85,B 0,C 180,E1 3412.139,E2 3412.139} C_VEL
LIN {X 0,Y 50.692,Z 1160.484,A -85,B 0,C 180,E1 3414.634,E2 3414.634} C_VEL
LIN {X 0,Y 41.484,Z 1162.088,A -85,B 0,C 180,E1 3416.279,E2 3416.279} C_VEL
LIN {X 0,Y 29.214,Z 1163.874,A -85,B 0,C 180,E1 3416.004,E2 3416.004} C_VEL
LIN {X 0,Y 7.481,Z 1165.957,A -85,B 0,C 180,E1 3402.466,E2 3402.466} C_VEL
LIN {X 0,Y 4.678,Z 1166.15,A -85,B 0,C 180,E1 3393.841,E2 3393.841} C_VEL
LIN {X 0,Y 6.871,Z 1166.955,A -85,B 0,C 180,E1 3241.825,E2 3241.825} C_VEL
LIN {X 0,Y 1.192,Z 1166.698,A -85,B 0,C 180,E1 3150.033,E2 3150.033} C_VEL
LIN {X 0,Y 16.205,Z 1165.24,A -85,B 0,C 180,E1 3050.813,E2 3050.813} C_VEL
LIN {X 0,Y 4.678,Z 1166.15,A -85,B 0,C 180,E1 3033.841,E2 3033.841} C_VEL
LIN {X 0,Y 3.022,Z 1168.145,A -85,B 0,C 180,E1 3020.866,E2 3020.866} C_VEL
LIN {X 0,Y 3.022,Z 1215,A -85,B 0,C 180,E1 3020.866,E2 3020.866} C_VEL
LIN {X 0,Y 3.022,Z 1215,A -85,B 0,C 180,E1 3020.866,E2 3020.866}

QRS_NEXT_CUT()

QRS_NEXT()
QRS_HOME()

END
